FUNCTION_BLOCK MACH_CTL (* Cycle Control for a Machine with Fixed Tool *)
  (* Standard: 61499-1; Classification: Simulation; ApplicationDomain: Machining; Function: Drilling *)
  (* Version 0.3, 2006-03-05, JHC, Holobloc Inc, Split SENSE int W_SENSE and M_SENSE; replaced ECC with directly invoked algorithms. *)
  (* Version 0.2, 2004-10-20, JHC, Rockwell Automation, Changed algorithm to LD to recover from retracting fault. *)
  (* Version 0.1, 2004-04-05, JHC, Rockwell Automation, Corrected transition SPIN -> ADV *)
  (* Version 0.0, 2002-10-03, JHC, Rockwell Automation, Modified from DRILL_CTL. *)
  (* Compiler header: package fb.rt.mach; *)
  (* Compiler Java Sun JDK 1.5.0 *)
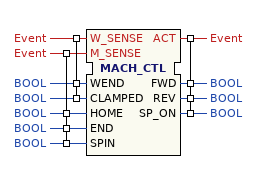
  EVENT_INPUT
    W_SENSE WITH WEND, CLAMPED; (* Workpiece Transport Sensors *)
    M_SENSE WITH END, SPIN, HOME; (* Machine Sensors *)
  END_EVENT
  EVENT_OUTPUT
    ACT WITH FWD, REV, SP_ON; (* Actuator output change *)
  END_EVENT
  VAR_INPUT
    WEND : BOOL; (* Workpiece present for machining *)
    CLAMPED : BOOL; (* Workpiece clamped *)
    HOME : BOOL; (* Machine home *)
    END : BOOL; (* Machine at END position *)
    SPIN : BOOL; (* Spindle at operating speed *)
  END_VAR
  VAR_OUTPUT
    FWD : BOOL; (* Advance machine *)
    REV : BOOL; (* Retract machine *)
    SP_ON : BOOL; (* Spindle motor *)
  END_VAR
  VAR
    MACHINED : BOOL; (* Machining operation completed on current piece *)
  END_VAR
  ALGORITHM W_SENSE IN ST: (* Workpiece sensor processing *)
SP_ON := CLAMPED;
MACHINED := MACHINED & WEND;
FWD := WEND & CLAMPED & SPIN & NOT END & NOT MACHINED;
REV := NOT FWD & NOT HOME;
ACT.serviceEvent(this);
  END_ALGORITHM
  ALGORITHM M_SENSE IN ST: (* Machine sensor processing *)
IF END & NOT MACHINED THEN
  MACHINED := TRUE;
  FWD := FALSE;
  REV := TRUE;
  ACT.serviceEvent(this);
ELSIF HOME & REV THEN
  REV := FALSE;
  ACT.serviceEvent(this);
ELSIF SPIN & WEND & CLAMPED & NOT END & NOT MACHINED & NOT FWD THEN
  FWD := TRUE;
  ACT.serviceEvent(this);
END_IF
  END_ALGORITHM
END_FUNCTION_BLOCK
